{attribute 'GeneratedUsingTerminal: KL8524'}
{attribute addProperty BoxType "KL8524"}
{attribute addProperty Id "StateAT %I*USINT0Auto_Manual_ChannelAT %I*BYTE0Switch_modeAT %I*BYTE0On_Off_ChannelAT %I*BYTE0CtrlAT %Q*USINT0Switch_mode_OutAT %Q*BYTE0Data_Reg_ComAT %Q*BYTE0LED_Out_greenAT %Q*BYTE0LED_Out_yellowAT %Q*BYTE0"}
{attribute addProperty CRC "845404373"}
{attribute addProperty Size "0"}
TYPE Channel_3263D8D5 :
STRUCT
	{attribute addProperty Name "State"}
	State AT %I* : USINT;
	{attribute addProperty Name "Auto_Manual_Channel"}
	Auto_Manual_Channel AT %I* : BYTE;
	{attribute addProperty Name "Switch_mode"}
	Switch_mode AT %I* : BYTE;
	{attribute addProperty Name "On_Off_Channel"}
	On_Off_Channel AT %I* : BYTE;
	{attribute addProperty Name "Ctrl"}
	Ctrl AT %Q* : USINT;
	{attribute addProperty Name "Switch_mode_Out"}
	Switch_mode_Out AT %Q* : BYTE;
	{attribute addProperty Name "Data_Reg_Com"}
	Data_Reg_Com AT %Q* : BYTE;
	{attribute addProperty Name "LED_Out_green"}
	LED_Out_green AT %Q* : BYTE;
	{attribute addProperty Name "LED_Out_yellow"}
	LED_Out_yellow AT %Q* : BYTE;
END_STRUCT
END_TYPE

(* stored: Version 1.2.0.0, ProductVersion 3.1.4024.9
   DUT Channel_3263D8D5: Id {f12d3a48-d300-4e99-b48f-0471d952b95c} *)
